KUKA KRL program: vw_Sto_cs_user.src, vw_Sto_cs_user.dat

--- vw_Sto_cs_user.src ---
&ACCESS RVEO
&REL 70
&PARAM DISKPATH = VW_User/Applikation/Vision/SMA
&PARAM TPVW_VERSION = 8.1.8
&PARAM EDITMASK = vw_cgx_user
DEF vw_sto_cs_user( )
;
;*---------------------------------------------*
;* Steinbichler Conzept Solutions GmbH             *
;* Version 1.0.0  / VKRC 4                               *
;* Bearbeitet am:                                          *
;* 20130208  vw_sto_cs_user erstellt                *
;*---------------------------------------------*
;
END
;
GLOBAL DEF STO_CS_Interface(USER_CMD :IN, CMD_SEL :IN,PAR1 :IN,PAR2 :IN, PAR3 :IN,PAR4 :IN,PAR5 :IN,PAR6 :IN)
  DECL VW_USER_CMD USER_CMD
  INT CMD_SEL,PAR1,PAR2,PAR3,PAR4,PAR5,PAR6

  SWITCH PAR1
  ;;FOLD VISIO7
  ;Start Integration VISIO7 durch CS JZ
  ;***********************************************
  ;
  ;***Legende***
	;PAR1 ==> Programmfunktion (1=Bewegung ausfuehren)
	;PAR2 ==> 1=pruefen ob Startpos == AxisRobGst(Home) / 2=nicht pruefen (aus Cell =>2 sonst 1)
	;PAR3 ==> Reserve
	;PAR4 ==> Reserve
	;PAR5 ==> Reserve
	;PAR6 ==> Reserve
	;**************
	;***Interrupts***
	; Interrupt 32 => NOT diZustimm , I_Zustimm()
	; Interrupt 33 => giZyklusCounterIn<>OldZyklusCounterIn , I_Multiplex()
	;**************

CASE 1 ;Bewegung von VISIO7 ausfuehren
 InitVisio () ;Variablen Initialisieren
 PTP $Pos_Act

 OldZyklusCounterIn=giZyklusCounterIn ;auf gleichen Wert setzen um Flanke fuer Interrupt zu bekommen
 INTERRUPT DECL 33 WHEN  giZyklusCounterIn<>OldZyklusCounterIn DO I_Multiplex()
 INTERRUPT ON 33 ;I_Multiplex
 WAIT FOR (OldZyklusCounterIn==giZyklusCounterIn) ; ;auf gleichen Wert warten um Flanke fuer Interrupt zu bekommen
 WAIT SEC 0.15 ;Wartezeit wegen Signalueberschneidung (Falnke Interrupt)
 OldZyklusCounterIn=0 ;mit 0 initialisieren

 IF (PAR2==1) THEN ;pruefen ob Startpos == AxisRobGst(Home)
  bRobGst=IN_AxPOS(AxisRobGst) ;Grundstellung Roboter pruefen Achswerte
  IF NOT bRobGst THEN ; Roboter nicht in Grundtstellung bei Programmeinsprung
   SetProgStatus(203) ;Programmstatus setzen (Legende im SetProgStatus)
   HALT ;ungueltige Startposition (nicht Home)
  ENDIF ; Roboter nicht in Grundtstellung bei Programmeinsprung
 ENDIF ;pruefen ob Startpos == AxisRobGst(Home)
  WAIT FOR bReadComplete ;eimal alle Daten eingelesen, da sonst kein Teachmode gesetzt ist und aus dem Programm gesprungen wird
   REPEAT  ;Onlinefahren ende
      WAIT SEC 0.1 ;Wartezeit wegen CPU-Auslastung
      SetProgStatus(0) ;Programmstatus setzen (Legende im SetProgStatus)

      IF bMoveToPos THEN
         GetSpeed() ;Geschwindigkeitsdaten aus XML auslesen
        IF bErrGetSpeed==FALSE THEN ;kein Fehler Speeddata
         GetPosition() ;Positionsdaten aus XML auslesen
        ENDIF
        bErrGetSpeed=FALSE ;Variable ruecksetzen
      ENDIF

    bRobGst=IN_AxPOS(AxisRobGst) ;Grundstellung Roboter pruefen Achswerte
    IF (bTeachMode==FALSE) AND (bRobGst==FALSE) THEN;teachen beendet, Rob aber nicht in Gst
     SetProgStatus(106) ;Programmstatus setzen (Legende im SetProgStatus)
    ENDIF ;teachen beendet, Rob aber nicht in Gst
   UNTIL (bTeachMode==FALSE) AND (bRobGst==TRUE) ;Onlinefahren ende

    PTP AxisRobGst ;AxisRobGst => entspricht Home in Config.dat
   WAIT SEC 0.0 ;Dummywartezeit wegen Vorlaufstop

   INTERRUPT OFF 33 ;I_Multiplex
    InitVisio () ;Variablen Initialisieren

   DEFAULT
  ENDSWITCH ;von PAR1
  ;***********************************************
  ;Ende Integration VISIO7 durch CS JZ
  ;lokale Unterprogramme am Schluss angehaengt
  ; => DEF InitVisio () ;Variablen Initialisieren
  ; => DEF SetProgStatus(Status :IN)
  ; => DEF GetPosition ()
  ; => DEF GetSpeed()
  ; => DEF MoveToPos()
  ; => DEF I_Zustimm()
  ; => DEF  I_Multiplex()
  ; => DEFFCT  BOOL IN_POS(CHECKPOS :IN)
  ; => DEFFCT  BOOL IN_AxPOS(CHECKPOS :IN)
  ; => DEFFCT INT ByteSwap(nInValue:IN, Lenght:IN, OutSequence:IN, DoFct:IN  )
  ;***********************************************
END
;-----------------------------------------------------------
DEF InitVisio () ;Variablen Initialisieren
 ;Variablen auf Startzuststand Initialisieren
 nProgStatus=0 ;Programmstatus ruecksetzen
 OldZyklusCounterIn=0 ;Multiplexvariable initialisiere
 goZyklusCounterOut=0 ;Ausgang Initialisieren
 bMoveToPos=FALSE ;Auf Position von Visio fahren
 bTeachMode=FALSE ;Teachmode aktiv
 bErrGetSpeed=FALSE ;Fehler in Geschwindigkeitsparameter
 $Timer[nLifeBitTimerNr]=nLifeBitTime ;Timer initialisieren
 $Timer_Stop[nLifeBitTimerNr]=TRUE ;Timer stoppen
 bReadComplete=FALSE ;Merker ruecksetzen
END
;-----------------------------------------------------------
DEF SetProgStatus(Status :IN)
;;FOLD SetProgStatus
   INT Status
   ;====== Legende  Programmstatus=======
   ; 0 => Ready
   ; 1 => Working
   ; 2 => ok (Befehl ausgefuerht)
   ; 10-99 => Zustand
   ; 10 => Robter wird gerade Handgefuehrt
   ;
   ; 100-999 => Fehler
   ; 100 =>
   ; 106 => Teachmode  beendet Roboter aber nicht in Home1 (Teachmode aktivieren undHome1 anfahren)
   ; 116 => anfahren des VisioPunkt durch loslassen der Zustimmtaste abgebrochen
   ; 117 => anfahren des VisioPunkt angewaehlt ohne Zustimmtaste
   ;
   ; 200 => Arbeitsraum-Fehler bei pPosVonVisio
   ; 201 => TURN-Fehler bei pPosVonVisio
   ; 202 => ungueltiger Geschwindigkeitsparameter
   ; 203 => Grundstellungspruefung bei Start TeachMode aktiv => Roboter aber nicht in GST
   ;
   ; 999 => schwerer Fehler Roboterpanel beachten
   ;================================

 IF bKommAktiv THEN ;wenn Kommunikation akitv ist
  WAIT FOR nProgStatusAck==nProgStatus ;Programmstatus Rueckmeldung von Visio
 ENDIF ;wenn Kommunikation akitv ist
 nProgStatus = Status ;Programmstatus setzen

;;ENDFOLD
END
;-----------------------------------------------------------
DEF GetPosition ()

;;FOLD GetPosition
   INTERRUPT DECL 32 WHEN NOT bZustimm DO I_Zustimm()

   IF bZustimm THEN ;wenn Zustimmtaste gedrueckt ist

   SetProgStatus(1) ;Programmstatus setzen (Legende im SetProgStatus)

   ;Positionsdaten wurden bereits im Multiplex-Programm gelesen
   ;Positionsdaten pruefen
   ;E6AXIS  INVERSE (E6POS  POSITION: IN, E6AXIS START_AXIS: IN,				 INT ERR_STATUS: OUT)
   ret=0 ;Variable initialisieren
   APOS1=INVERSE(pPosVonVisio,$Axis_Act,ret)
   IF ret<>0 THEN
    IF ret==2 THEN ;2Arbeitsraum-Fehler bei der math. Trafo-Funktion, d.h. es gibt keine Achswinkel, mit denen die kartesische Zielposition erreicht werden kann
     SetProgStatus(200) ;Programmstatus setzen (Legende im SetProgStatus)
     ELSE ;2
      IF ret==3 THEN ;3 Es gibt zwar Loesungswinkel, aber mit dem gegebenem Turn werden SW-Endschalter verletzt
       SetProgStatus(201) ;Programmstatus setzen (Legende im SetProgStatus)
       ELSE ;3
         HALT ;Roboterposition nicht erreichbar
      ENDIF ;3
    ENDIF ;2
   ELSE ;<>0
   MoveToPos() ;Position anfahren
   ENDIF ;<>0

  ELSE ;wenn Zustimmtaste gedrueckt ist
   SetProgStatus(117) ;Position anfahren gewaehlt aber Zustimmtaste nicht gedrueckt
  ENDIF ;wenn Zustimmtaste gedrueckt ist

;;ENDFOLD
END
;-----------------------------------------------------------
DEF GetSpeed()
;   ;FOLD GetSpeed
   INT Factor,I

   bErrGetSpeed=FALSE ;Variable ruecksetzen

   ; $APO.CDIS
   IF (TeachSpeed.ApoCdis>0) AND (TeachSpeed.ApoCdis<=200) THEN
    IF TeachSpeed.ApoCdis>SpeedLimit.ApoCdis THEN
     TeachSpeed.ApoCdis=SpeedLimit.ApoCdis
    ENDIF
    $APO.CDIS=TeachSpeed.ApoCdis
   ELSE
    SetProgStatus(202) ;Programmstatus setzen (Legende im SetProgStatus)
    User_Msg(2) ;Meldungsausgabe am KCP
    bErrGetSpeed=TRUE ;Variable setzen
   ENDIF

   ; $VEL.CP
   IF (TeachSpeed.VelCp>0) AND (TeachSpeed.VelCp<=2.0) THEN
    IF TeachSpeed.VelCp>SpeedLimit.VelCp THEN
     TeachSpeed.VelCp=SpeedLimit.VelCp
    ENDIF
    $VEL.CP=TeachSpeed.VelCp
   ELSE
    SetProgStatus(202) ;Programmstatus setzen (Legende im SetProgStatus)
    User_Msg(3) ;Meldungsausgabe am KCP
    bErrGetSpeed=TRUE ;Variable setzen
   ENDIF

   ; $ACC.CP
   IF (TeachSpeed.AccCp>0) AND (TeachSpeed.AccCp<=2.3) THEN
    IF TeachSpeed.AccCp>SpeedLimit.AccCp THEN
     TeachSpeed.AccCp=SpeedLimit.AccCp
    ENDIF
    $ACC.CP=TeachSpeed.AccCp
   ELSE
    SetProgStatus(202) ;Programmstatus setzen (Legende im SetProgStatus)
    User_Msg(4) ;Meldungsausgabe am KCP
    bErrGetSpeed=TRUE ;Variable setzen
   ENDIF

   ; $VEL.ORI2
   IF (TeachSpeed.VelOri>0) AND (TeachSpeed.VelOri<=200.0) THEN
    IF TeachSpeed.VelOri>SpeedLimit.VelOri THEN
     TeachSpeed.VelOri=SpeedLimit.VelOri
    ENDIF
    $VEL.ORI1=TeachSpeed.VelOri
    $VEL.ORI2=TeachSpeed.VelOri
   ELSE
    SetProgStatus(202) ;Programmstatus setzen (Legende im SetProgStatus)
    User_Msg(5) ;Meldungsausgabe am KCP
    bErrGetSpeed=TRUE ;Variable setzen
   ENDIF

   ; VELPTP
   ;Factor darf zwischen 0 und 100 liegen
   IF TeachSpeed.VelPtp>SpeedLimit.VelPtp THEN
      TeachSpeed.VelPtp=SpeedLimit.VelPtp
      IF bStopOnError THEN ;bei Fehler halten
       HALT
      ENDIF ;bei Fehler halten
   ENDIF
   IF TeachSpeed.VelPtp<1 THEN ;min 1% Geschwindigkeit
      TeachSpeed.VelPtp=1
      IF bStopOnError THEN ;bei Fehler halten
       HALT
      ENDIF ;bei Fehler halten
   ENDIF
   ;Achsgeschwindigkeiten setzen
   FOR I=1 TO $NUM_AX
      $VEL_AXIS[I]=TeachSpeed.VelPtp
   ENDFOR

   ; ACCPTP
   ;Factor darf zwischen 0 und 100 liegen
   IF TeachSpeed.AccPtp>SpeedLimit.AccPtp THEN
      TeachSpeed.AccPtp=SpeedLimit.AccPtp
   ENDIF
   IF TeachSpeed.AccPtp<1 THEN ;min 1% Beschleunigung
      TeachSpeed.AccPtp=1
   ENDIF
   ;Achsgeschwindigkeiten setzen
   FOR I=1 TO $NUM_AX
      $ACC_AXIS[I]=TeachSpeed.AccPtp
   ENDFOR

   ; $VEL_EXTAX[1]
   ;Factor darf zwischen 0 und 100 liegen
   IF TeachSpeed.VelExtAx1>SpeedLimit.VelExtAx1 THEN
      TeachSpeed.VelExtAx1=SpeedLimit.VelExtAx1
   ENDIF
   IF TeachSpeed.VelExtAx1<1 THEN ;min 1%
      TeachSpeed.VelExtAx1=1
   ENDIF
   ;Achsgeschwindigkeiten setzen
   $VEL_EXTAX[1]=TeachSpeed.VelExtAx1

   ; $VEL_EXTAX[2]
   ;Factor darf zwischen 0 und 100 liegen
   IF TeachSpeed.VelExtAx2>SpeedLimit.VelExtAx2 THEN
      TeachSpeed.VelExtAx2=SpeedLimit.VelExtax2
   ENDIF
   IF TeachSpeed.VelExtAx2<1 THEN ;min 1%
      TeachSpeed.VelExtAx2=1
   ENDIF
   ;Achsgeschwindigkeiten setzen
   $VEL_EXTAX[2]=TeachSpeed.VelExtAx2

;;ENDFOLD
END
;-----------------------------------------------------------
DEF MoveToPos()
   INTERRUPT ON 32 ;Bewegung abbrechen
   WAIT FOR bZustimm ;Zustimmstaste gedrueckt
   IF bMovePTP THEN ;Bewegung ist PTP
      PTP pPosVonVisio ;Punkt anfahren
   ELSE
      LIN pPosVonVisio ;Punkt anfahren
   ENDIF
   Interrupt OFF 32 ;Bewegung abbrechen
   SetProgStatus(2) ;Programmstatus setzen (Legende im SetProgStatus)
END
;-----------------------------------------------------------
DEF I_Zustimm()
   Interrupt OFF 32 ;Bewegung abbrechen
   Brake ;Roboter anhalten
   SetProgStatus(116) ;Programmstatus setzen (Legende im SetProgStatus)
   Resume ;Ruecksprung ins Hauptprogramm
END
;-----------------------------------------------------------
DEF I_Multiplex()
;20130121 JZ => erstellt
;20130125 JZ => neue Signalliste verwendet, Shattendaten erstellt
;29130125 JZ => in VW_USR_R integriert

;bei 5 auf 0 Ruecksetzen, wegen Errorflag bei verpassten Paketen
IF (OldZyklusCounterIn==MultiplexFaktor) OR  ($Timer_Flag[nLifeBitTimerNr]) THEN
 OldZyklusCounterIn=0
 IF $Timer_Flag[nLifeBitTimerNr] THEN
  $Timer[nLifeBitTimerNr]=nLifeBitTime ;Timer initialisieren
  $Timer_Stop[nLifeBitTimerNr]=FALSE ;Timer starten
 ENDIF
ENDIF

IF (ErrorFlag==FALSE) AND (giZyklusCounterIn>1)  AND (giZyklusCounterIn-OldZyklusCounterIn >1) THEN ;Paketverlust
 ErrorFlag=TRUE ;Fehler
 ErrorCounter=ErrorCounter+1 ;Fehlerzaehler hochzaehlen
ENDIF ;Paketverlust

OldZyklusCounterIn=giZyklusCounterIn ;Merker setzen

IF goZyklusCounterOut==giZyklusCounterOutAck THEN ;Im Handhakemodus auf Bestaetigung ZyklusCounterOut warten
goZyklusCounterOut=goZyklusCounterOut+1 ;hochzaehlen
 IF (goZyklusCounterOut>MultiplexFaktor) THEN
  goZyklusCounterOut=1 ;ruecksetzen
 ENDIF
ENDIF

;Am Anfang einer Runde die Schattendaten schreiben
IF goZyklusCounterOut==1 THEN
 ;allgemeine Daten in Schattendaten schreiben
 bSdwDoLifeBit=bLifeBitOld ;
 bSdwDoStopMess=$StopMess ;
 nSdwGoProgStatus=nProgStatus
 nSdwGoRobTimer=$Rob_Timer
 nSdwGoFloatFaktor=nFloatFaktor*10
 ;Positionsdaten in Schattendaten schreiben
 pShadowPosAnVisio=$Pos_Act ;aktuelle Position in Schattendaten speichern
ENDIF

;eine Seite einlesen
IF (giZyklusCounterIn>=1) AND (giZyklusCounterIn<= MultiplexFaktor) THEN
 IF giZyklusCounterIn==1 THEN ;allgemeine Daten
  bSdwDiKommAktiv=diKommAtiv ;
  bSdwDiTeachMode=diTeachMode ;
  bSdwDiMovePTP=diMovePTP ;
  bSdwDiMoveToPos=diMoveToPos ;
  bSdwDiLifeBit=diLifeBit ;
  nSdwGiProgStatusAck=ByteSwap(giProgStatusAck, 16, 21, TRUE) ;
  nSdwGiFloatFaktor=giFloatFaktor*10 ;
  IF nSdwGiFloatFaktor==0 THEN ;ungueltiger Wert wegen Division durch Null
   nSdwGiFloatFaktor=1 ;Wert initialisieren
  ENDIF
 ENDIF ;allgemeine Daten
 IF giZyklusCounterIn==2 THEN ;X/Y/Z
  IF nSdwGiFloatFaktor==0 THEN ;ungueltiger Wert wegen Division durch Null
   nSdwGiFloatFaktor=1 ;Wert initialisieren
  ENDIF
  pShadowPosVonVisio.X=ByteSwap(giPosX, 32, 4321, TRUE)/nSdwGiFloatFaktor
  pShadowPosVonVisio.Y=ByteSwap(giPosY, 32, 4321, TRUE)/nSdwGiFloatFaktor
  pShadowPosVonVisio.Z=ByteSwap(giPosZ, 32, 4321, TRUE)/nSdwGiFloatFaktor
 ENDIF ;X/Y/Z
 IF giZyklusCounterIn==3 THEN ;A/B/C
  IF nSdwGiFloatFaktor==0 THEN ;ungueltiger Wert wegen Division durch Null
   nSdwGiFloatFaktor=1 ;Wert initialisieren
  ENDIF
  pShadowPosVonVisio.A=ByteSwap(giPosA, 32, 4321, TRUE)/nSdwGiFloatFaktor
  pShadowPosVonVisio.B=ByteSwap(giPosB, 32, 4321, TRUE)/nSdwGiFloatFaktor
  pShadowPosVonVisio.C=ByteSwap(giPosC, 32, 4321, TRUE)/nSdwGiFloatFaktor
 ENDIF ;A/B/C
 IF giZyklusCounterIn==4 THEN ;E1/E2/S/T
  IF nSdwGiFloatFaktor==0 THEN ;ungueltiger Wert wegen Division durch Null
   nSdwGiFloatFaktor=1 ;Wert initialisieren
  ENDIF
  pShadowPosVonVisio.E1=ByteSwap(giPosE1, 32, 4321, TRUE)/nSdwGiFloatFaktor
  pShadowPosVonVisio.E2=ByteSwap(giPosE2, 32, 4321, TRUE)/nSdwGiFloatFaktor
  pShadowPosVonVisio.S=giPosS
  pShadowPosVonVisio.T=giPosT ;ByteSwap???
 ENDIF ;E1/E2/S/T
 IF giZyklusCounterIn==5 THEN ;Geschwindigkeitsdaten
  IF nSdwGiFloatFaktor==0 THEN ;ungueltiger Wert wegen Division durch Null
   nSdwGiFloatFaktor=1 ;Wert initialisieren
  ENDIF
  SdwTeachSpeed.ApoCdis=ByteSwap(giApoCdis, 16, 21, TRUE)/100.0
  SdwTeachSpeed.VelCp=ByteSwap(giVelCp, 16, 21, TRUE)/1000.0
  SdwTeachSpeed.AccCp=ByteSwap(giAccCp, 16, 21, TRUE)/100.0
  SdwTeachSpeed.VelOri=ByteSwap(giVelOri, 16, 21, TRUE)
  SdwTeachSpeed.VelPtp=giVelPtp
  SdwTeachSpeed.AccPtp=giAccPtp
  SdwTeachSpeed.VelExtAx1=giVelExtAx1
  SdwTeachSpeed.VelExtAx2=giVelExtAx2
 ENDIF ;Geschwindigkeitsdaten
ENDIF

;eine Seite schreiben
IF (goZyklusCounterOut>=1) AND (goZyklusCounterOut<=MultiplexFaktor) THEN
 IF goZyklusCounterOut==1 THEN ;allgemeine Daten
  I4=$Rob_timer-I3 ;IBN
  I3=$Rob_timer ;IBN
  doLifeBit=bSdwDoLifeBit
  doStopMess=bSdwDoStopMess
  goProgStatus=ByteSwap(nSdwGoProgStatus, 16, 21, TRUE)
  goRobTimer=ByteSwap(nSdwGoRobTimer, 32, 4321, TRUE)
  goFloatFaktor=nSdwGoFloatFaktor/10
 ENDIF ;allgemeine Daten
 IF goZyklusCounterOut==2 THEN ;X/Y/Z
  goPosX=ByteSwap((pShadowPosAnVisio.X*nSdwGoFloatFaktor), 32, 4321, TRUE)
  goPosY=ByteSwap((pShadowPosAnVisio.Y*nSdwGoFloatFaktor), 32, 4321, TRUE)
  goPosZ=ByteSwap((pShadowPosAnVisio.Z*nSdwGoFloatFaktor), 32, 4321, TRUE)
  nGoPosX=goPosX ;IBN
  nGoPosY=goPosY ;IBN
  nGoPosZ=goPosZ ;IBN
 ENDIF ;X/Y/Z
 IF goZyklusCounterOut==3 THEN ;A/B/C
  goPosA=ByteSwap((pShadowPosAnVisio.A*nSdwGoFloatFaktor), 32, 4321, TRUE)
  goPosB=ByteSwap((pShadowPosAnVisio.B*nSdwGoFloatFaktor), 32, 4321, TRUE)
  goPosC=ByteSwap((pShadowPosAnVisio.C*nSdwGoFloatFaktor), 32, 4321, TRUE)
  nGoPosA=goPosA ;IBN
  nGoPosB=goPosB ;IBN
  nGoPosC=goPosC ;IBN
 ENDIF ;A/B/C
 IF goZyklusCounterOut==4 THEN ;E1/E2/S/T
  goPosE1=ByteSwap((pShadowPosAnVisio.E1*nSdwGoFloatFaktor), 32, 4321, TRUE)
  goPosE2=ByteSwap((pShadowPosAnVisio.E2*nSdwGoFloatFaktor), 32, 4321, TRUE)
  goPosS=pShadowPosAnVisio.S
  goPosT=pShadowPosAnVisio.T
  goPosT2=0 ;ReserveTurn auf 0 initialisieren
  goPosT3=0 ;ReserveTurn auf 0 initialisieren
  nGoPosE1=goPosE1 ;IBN
  nGoPosE2=goPosE2 ;IBN
  nGoPosS=goPosS ;IBN
  nGoPosT=goPosT ;IBN
 ENDIF ;E1/E2/S/T
 IF goZyklusCounterOut==5 THEN ;Reserve
  ;nicht belegt
 ENDIF ;
ENDIF

;Am Ende einer Runde die Schattendaten uebernehmen
IF (ErrorFlag==FALSE) AND (giZyklusCounterIn==MultiplexFaktor) THEN
  bKommAktiv=bSdwDiKommAktiv ;
  bTeachMode=bSdwDiTeachMode ;
  bMovePTP=bSdwDiMovePTP ;
  bMoveToPos=bSdwDiMoveToPos ;
  bLifeBit=bSdwDiLifeBit ;
  nProgStatusAck=nSdwGiProgStatusAck ;
  ;nSdwGiFloatFaktor ;wird nur im Multiplexbereich benoetigt
  pPosVonVisio=pShadowPosVonVisio ;Positionsdaten uebergeben
  TeachSpeed.ApoCdis =SdwTeachSpeed.ApoCdis
  TeachSpeed.VelCp =SdwTeachSpeed.VelCp
  TeachSpeed.AccPtp =SdwTeachSpeed.AccPtp
  TeachSpeed.VelOri =SdwTeachSpeed.VelOri
  TeachSpeed.VelPtp =SdwTeachSpeed.VelPtp
  TeachSpeed.AccPtp =SdwTeachSpeed.AccPtp
  TeachSpeed.VelExtAx1 =SdwTeachSpeed.VelExtAx1
  TeachSpeed.VelExtAx2 =SdwTeachSpeed.VelExtAx2
  ;Lifebit
  IF bLifeBit==bLifeBitOld THEN ;LifeBit vergleichen
   bLifeBitOld=NOT bLifeBitOld ;Lifebit negieren
   I2=$Rob_timer-I1 ;IBN
   I1=$Rob_timer ;IBN
   $Timer[nLifeBitTimerNr]=nLifeBitTime ;Timer initialisieren
   $Timer_Stop[nLifeBitTimerNr]=FALSE ;Timer starten
  ENDIF ;LifeBit vergleichen
 bReadComplete=TRUE ;1 Datensatz komplett gelesen
ENDIF

IF ErrorFlag AND (giZyklusCounterIn==1) THEN
 ErrorFlag=FALSE ;Flag ruecksetzen
ENDIF

;Spiegeln fuer die Gegenseite
goZyklusCounterInAck=giZyklusCounterIn

END
;-----------------------------------------------------------
;FOLD Position pruefen
DEFFCT  BOOL IN_POS(CHECKPOS :IN)
DECL E6POS CHECKPOS
DECL BOOL B_IN_POS
B_IN_POS=TRUE
IF (CHECKPOS.X<$POS_ACT.X-TolTrans) OR (CHECKPOS.X>$POS_ACT.X+TolTrans) THEN
 B_IN_POS=FALSE
ENDIF
IF (CHECKPOS.Y<$POS_ACT.Y-TolTrans) OR (CHECKPOS.Y>$POS_ACT.Y+TolTrans) THEN
 B_IN_POS=FALSE
ENDIF
IF (CHECKPOS.Z<$POS_ACT.Z-TolTrans) OR (CHECKPOS.Z>$POS_ACT.Z+TolTrans) THEN
 B_IN_POS=FALSE
ENDIF
IF (CHECKPOS.A<$POS_ACT.A-TolRot) OR (CHECKPOS.A>$POS_ACT.A+TolRot) THEN
 B_IN_POS=FALSE
ENDIF
IF (CHECKPOS.B<$POS_ACT.B-TolRot) OR (CHECKPOS.B>$POS_ACT.B+TolRot) THEN
 B_IN_POS=FALSE
ENDIF
IF (CHECKPOS.C<$POS_ACT.C-TolRot) OR (CHECKPOS.C>$POS_ACT.C+TolRot) THEN
 B_IN_POS=FALSE
ENDIF
IF (CHECKPOS.E1<$POS_ACT.E1-TolRot) OR (CHECKPOS.E1>$POS_ACT.E1+TolRot) THEN
 B_IN_POS=FALSE
ENDIF
IF (CHECKPOS.E2<$POS_ACT.E2-TolRot) OR (CHECKPOS.E2>$POS_ACT.E2+TolRot) THEN
 B_IN_POS=FALSE
ENDIF
RETURN  (B_IN_POS)
ENDFCT ;Function IN_POS
;ENDFOLD
;-----------------------------------------------------------
;FOLD Achsposition pruefen
DEFFCT  BOOL IN_AxPOS(CHECKPOS :IN)
DECL E6AXIS CHECKPOS
DECL BOOL B_IN_POS
B_IN_POS=TRUE
IF (CHECKPOS.A1<$AXIS_ACT.A1-TolRot) OR (CHECKPOS.A1>$AXIS_ACT.A1+TolRot) THEN
 B_IN_POS=FALSE
ENDIF
IF (CHECKPOS.A2<$AXIS_ACT.A2-TolRot) OR (CHECKPOS.A2>$AXIS_ACT.A2+TolRot) THEN
 B_IN_POS=FALSE
ENDIF
IF (CHECKPOS.A3<$AXIS_ACT.A3-TolRot) OR (CHECKPOS.A3>$AXIS_ACT.A3+TolRot) THEN
 B_IN_POS=FALSE
ENDIF
IF (CHECKPOS.A4<$AXIS_ACT.A4-TolRot) OR (CHECKPOS.A4>$AXIS_ACT.A4+TolRot) THEN
 B_IN_POS=FALSE
ENDIF
IF (CHECKPOS.A5<$AXIS_ACT.A5-TolRot) OR (CHECKPOS.A5>$AXIS_ACT.A5+TolRot) THEN
 B_IN_POS=FALSE
ENDIF
IF (CHECKPOS.A6<$AXIS_ACT.A6-TolRot) OR (CHECKPOS.A6>$AXIS_ACT.A6+TolRot) THEN
 B_IN_POS=FALSE
ENDIF
IF (CHECKPOS.E1<$AXIS_ACT.E1-TolRot) OR (CHECKPOS.E1>$AXIS_ACT.E1+TolRot) THEN
 B_IN_POS=FALSE
ENDIF
IF (CHECKPOS.E2<$AXIS_ACT.E2-TolRot) OR (CHECKPOS.E2>$AXIS_ACT.E2+TolRot) THEN
 B_IN_POS=FALSE
ENDIF
RETURN  (B_IN_POS)
ENDFCT ;Function IN_POS
;ENDFOLD
;-----------------------------------------------------------
DEFFCT INT ByteSwap(nInValue:IN, Lenght:IN, OutSequence:IN, DoFct:IN  )

INT Result ;Ergebnis der Funktion
INT nInValue ;Eingangswert der umgewandelt werden soll
INT Lenght ;Bitanzahl des Eingangswertes (16 / 32)
BOOL DoFct ;ob die Funktion ausgefuehrt werden soll
INT SwapByte1, SwapByte2, SwapByte3, SwapByte4 ;Rechenbytes
INT OutSequence ;Reihenfolge in der die Bytes ausgegeben werden (z.B. Eingang 1,2,3,4 => Ausgang 4,3,2,1)
BOOL HiBit ;fuer Auswertung negative Zahl

;#######################################
;Wenn allgemein diese Funktion ausgeschaltet werden soll hier die Variable setzen
;DoFct=FALSE
;#######################################

IF DoFct THEN ;Berechnungen ausfuehren
 SwapByte1='B00000000' ;Initialisieren
 SwapByte2='B00000000' ;Initialisieren
 SwapByte3='B00000000' ;Initialisieren
 SwapByte4='B00000000' ;Initialisieren
 SWITCH Lenght
 ;----------------------------------------
  CASE 16 ;16 Bit Eingang
   SWITCH OutSequence ;Reihenfolge der Bytes
   ;==================================
    CASE 21
     SwapByte1= nInValue B_AND 'B1111111100000000'
     SwapByte2= nInValue B_AND 'B0000000011111111'
     SwapByte1=SwapByte1/256 ;Byte um 1 nach hinten schieben (2=>1)
     SwapByte2=SwapByte2*256 ;Byte um 1 nach vorn schieben (1=>2)
     Result=SwapByte1+SwapByte2 ;SwapBytes addieren
   ;==================================
    DEFAULT ;Reihenfolge der Bytes
     User_Msg(6) ;Meldungsausgabe am KCP
    ENDSWITCH ;Reihenfolge der Bytes
 ;----------------------------------------
  CASE 32 ;32 Bit Eingang
   SWITCH OutSequence ;Reihenfolge der Bytes
   ;==================================
    CASE 4321
     SwapByte1= nInValue B_AND 'B01111111000000000000000000000000'
     HiBit = (nInValue B_AND 'B10000000000000000000000000000000' <>0) ;abfangen wegen Negativer Zahlen (an Ende +128 rechnen)
     SwapByte2= nInValue B_AND 'B00000000111111110000000000000000'
     SwapByte3= nInValue B_AND 'B00000000000000001111111100000000'
     SwapByte4= nInValue B_AND 'B00000000000000000000000011111111'
     SwapByte1=(((SwapByte1/256)/256)/256) ;Byte um 3 nach hinten schieben (4=>1)
     SwapByte2=SwapByte2/256 ;Byte um 1 nach hinten schieben (3=>2)
     SwapByte3=SwapByte3*256 ;Byte um 1 nach vorn schieben (2=>3)
     SwapByte4=(((SwapByte4*256)*256)*256) ;Byte um 3 nach vorn schieben (1=>4)
     IF HiBit THEN
      Result=SwapByte1+SwapByte2+SwapByte3+SwapByte4+128 ;SwapBytes addieren und 128 hinzuzaehlen wegen Negativzahl
     ELSE
      Result=SwapByte1+SwapByte2+SwapByte3+SwapByte4 ;SwapBytes addieren
     ENDIF
   ;==================================
    DEFAULT ;Reihenfolge der Bytes
     User_Msg(7) ;Meldungsausgabe am KCP
    ENDSWITCH ;Reihenfolge der Bytes
 ;----------------------------------------
  DEFAULT ;BitZahl
   User_Msg(8) ;Meldungsausgabe am KCP
 ENDSWITCH ;BitZahl

ELSE ;Berechnungen ausfuehren
 Result=nInValue ;Rueckgabewert aus Eingabewert setzen bei Nichtberechnung
ENDIF  ;Berechnungen ausfuehren

RETURN(Result) ;Ergebnis von Funktion Uebergeben
ENDFCT

;-----------------------------------------------------------
DEF User_Msg(MyMsgNr:IN )

 ;FOLD Versionslegende

 ;ENDFOLD
;aktuelle Version: V1.0

DECL KrlMsg_T My_Meldung
DECL KrlMsgPar_T My_Parameter[3]
DECL KrlMsgOpt_T My_Option
DECL KrlMsgDlgSK_T My_SK[7]
int Result, MyMsgNr, Answer
;BOOL Clear_Ok ;Global in $Config.dat
INT MsgHandle[200] ;Handle der Meldung

;---------------------------------------------------
;#notify => Hinweismeldung
;                 -(nur mit Quitt / Alles Quitt)
;#state => Zustandsmeldung
;                -(von Programm aus löschbar)
;#quit => Quittiermeldung
;              -(Quitt / Alles Quitt mit rueckmeldung zum Programm)
;#waiting => Wartemeldung
;                  -(Simuliere oder auf Programmbedingung warten)
;---------------------------------------------------

;alle Mledungen loeschen
;Clear_OK = Clear_KrlMsg(-99) ; Meldungen im Puffer zurueck nehmen
IF bShowUserMsg THEN ;Meldungen anzeigen
SWITCH MyMsgNr
;---------------------------------------------------
 CASE 1 ;
  My_Meldung = {Modul[] "STO-CS", Nr 000, Msg_txt[] "fehlerhafte Gruppennummer uebergeben"}
  My_Meldung.Nr = MyMsgNr
  My_Option = {VL_Stop True, Clear_P_Reset True, Log_To_DB True}
  MsgHandle[MyMsgNr] = Set_KrlMsg(#state, My_Meldung, My_Parameter[], My_Option)
;---------------------------------------------------
 CASE 2 ;
  My_Meldung = {Modul[] "STO-CS", Nr 000, Msg_txt[] "TeachSpeed.ApoCdis => Wert ungueltig"}
  My_Meldung.Nr = MyMsgNr
  My_Option = {VL_Stop True, Clear_P_Reset True, Log_To_DB True}
  MsgHandle[MyMsgNr] = Set_KrlMsg(#state, My_Meldung, My_Parameter[], My_Option)
;---------------------------------------------------
 CASE 3 ;
  My_Meldung = {Modul[] "STO-CS", Nr 000, Msg_txt[] "TeachSpeed.VelCp => Wert ungueltig"}
  My_Meldung.Nr = MyMsgNr
  My_Option = {VL_Stop True, Clear_P_Reset True, Log_To_DB True}
  MsgHandle[MyMsgNr] = Set_KrlMsg(#state, My_Meldung, My_Parameter[], My_Option)
;---------------------------------------------------
 CASE 4 ;
  My_Meldung = {Modul[] "STO-CS", Nr 000, Msg_txt[] "TeachSpeed.AccCp => Wert ungueltig"}
  My_Meldung.Nr = MyMsgNr
  My_Option = {VL_Stop True, Clear_P_Reset True, Log_To_DB True}
  MsgHandle[MyMsgNr] = Set_KrlMsg(#state, My_Meldung, My_Parameter[], My_Option)
;---------------------------------------------------
 CASE 5 ;
  My_Meldung = {Modul[] "STO-CS", Nr 000, Msg_txt[] "TeachSpeed.VelOri => Wert ungueltig"}
  My_Meldung.Nr = MyMsgNr
  My_Option = {VL_Stop True, Clear_P_Reset True, Log_To_DB True}
  MsgHandle[MyMsgNr] = Set_KrlMsg(#state, My_Meldung, My_Parameter[], My_Option)
;---------------------------------------------------
 CASE 6 ;
  My_Meldung = {Modul[] "STO-CS", Nr 000, Msg_txt[] "OutSequence 16Bit Eingabe ByteSwap nicht definiert!"}
  My_Meldung.Nr = MyMsgNr
  My_Option = {VL_Stop True, Clear_P_Reset True, Log_To_DB True}
  MsgHandle[MyMsgNr] = Set_KrlMsg(#state, My_Meldung, My_Parameter[], My_Option)
;---------------------------------------------------
 CASE 7 ;
  My_Meldung = {Modul[] "STO-CS", Nr 000, Msg_txt[] "OutSequence 32Bit Eingabe ByteSwap nicht definiert!"}
  My_Meldung.Nr = MyMsgNr
  My_Option = {VL_Stop True, Clear_P_Reset True, Log_To_DB True}
  MsgHandle[MyMsgNr] = Set_KrlMsg(#state, My_Meldung, My_Parameter[], My_Option)
;---------------------------------------------------
 CASE 8 ;
  My_Meldung = {Modul[] "STO-CS", Nr 000, Msg_txt[] "Eingabe Bitlaenge ByteSwap unbekannt!"}
  My_Meldung.Nr = MyMsgNr
  My_Option = {VL_Stop True, Clear_P_Reset True, Log_To_DB True}
  MsgHandle[MyMsgNr] = Set_KrlMsg(#state, My_Meldung, My_Parameter[], My_Option)
;---------------------------------------------------
	CASE 151 ;
		My_Meldung = {Modul[] "STO-CS", Nr 000, Msg_txt[] "Teachmode beendet, Teachmode aktivieren und Roboter in Grundstellung bringen"}
    My_Meldung.Nr = MyMsgNr
		My_Option = {VL_Stop True, Clear_P_Reset True, Clear_P_SAW True, Log_To_DB False}
		MsgHandle[MyMsgNr] = Set_KrlMsg(#Quit, My_Meldung, My_Parameter[], My_Option)
	 WHILE (Exists_KrlMsg(MsgHandle[MyMsgNr])) ;warten bis der Anwender quittiert hat
			WAIT SEC 0.1
		ENDWHILE
	;---------------------------------------------------
DEFAULT
  My_Meldung = {Modul[] "STO-CS", Nr 000, Msg_txt[] "kein Meldetext vorhanden"}
  My_Meldung.Nr = MyMsgNr
  My_Option = {VL_Stop True, Clear_P_Reset True, Log_To_DB False}
  MsgHandle[MyMsgNr] = Set_KrlMsg(#State, My_Meldung, My_Parameter[], My_Option)
		WHILE (Exists_KrlMsg(MsgHandle[MyMsgNr])) ;warten bis der Anwender quittiert hat
			WAIT SEC 0.1
		ENDWHILE
  ;WAIT FOR FALSE
ENDSWITCH
ENDIF ;Meldungen anzeigen

END
;-----------------------------------------------------------
GLOBAL DEF STO_CS_SPS ()
;*** Zusatz für Teachmode mit VISIO7 (CS JZ) ***
 IF $Timer_Flag[nLifeBitTimerNr] THEN ;Timeout Lifebit
  bZustimm=FALSE ;Zustimmtaste ruecksetzen um Bewegung anzubrechen
 ELSE ;kein TimeOut
  bZustimm=diZustimm ;Uebergabe, da bei Busfehler und anstehendem Signal trotzdem gestoppt werden soll
 ENDIF ;Timeout LifeBit
;*** ENDE ****
END

--- vw_Sto_cs_user.dat ---
&ACCESS  RV
&PARAM DISKPATH = VW_User/Applikation/Vision/SMA
&PARAM EDITMASK = vw_cgx_user
&PARAM TPVW_VERSION = 8.1.8
&REL 69
DEFDAT  vw_Sto_cs_user PUBLIC
;
;FOLD STO_CS
;
;*---------------------------------------------*
;* Steinbichler CS GmbH                        *
;*                                             *
;* Bearbeitet am:                              *
;* 20130208 JZ                                 *
;*     vw_sto_cs_user  erstellt                *
;* 20151219 MBA                                *
;*     b_zustimm entfernt                      *
;*---------------------------------------------*
;
GLOBAL BOOL B_MIT_STO_CS=TRUE

INT I1=10717152
INT I2=3311112
INT I3=10721412
INT I4=88

;Allgemeine Variablen
BOOL bReadComplete=FALSE ;Merker 1 Zyklus komplett gelesen
;BOOL bErrGetSpeed=FALSE ;Fehler in Geschwindigkeitsparameter
BOOL bKommAktiv=FALSE ;Kommunikation mit Visio7 aktiv
BOOL bMoveToPos=FALSE ;Auf Position von Visio fahren
INT nProgStatusAck=0 ;Quittierung Programmstatus von Visio
INT nProgStatus=0 ;aktueller Programmstatus
;INT nRobTimer=0 ;Timestamp 1Inc=2ms
;in Config.dat ;BOOL bZustimm=TRUE ;Zustimmtaste
BOOL bMovePTP=FALSE ;Bewegung als PTP(TRUE) oder LIN(FALSE) ausfuehren
BOOL bTeachMode=FALSE ;Teachmode aktiv
BOOL bLifeBit=FALSE ;Lifebit zu Visio7
BOOL bLifeBitOld=TRUE ;Lifebit zu Visio7
GLOBAL BOOL bShowUserMsg=TRUE ;Meldungen am KCP anzeigen

;Allgemeine E/A
DECL E6AXIS APOS1={A1 8.13010216,A2 -82.4998856,A3 76.0127487,A4 269.075317,A5 98.0776978,A6 83.4475708,E1 0.0,E2 0.0,E3 0.0,E4 0.0,E5 0.0,E6 0.0} ;Achspos pPosVonVosio nach Inverse
;DECL E6AXIS APOS1={A1 0.969305158,A2 -145.691193,A3 140.448578,A4 -0.00214473042,A5 -106.031944,A6 -0.756430626,E1 0.000104831379,E2 0.000104831379,E3 0.0,E4 0.0,E5 0.0,E6 0.0} ;Achspos pPosVonVosio nach Inverse
INT ret=0 ;Returnwert aus Inverse-Funktion zur kontrolle ob pPosVonVisio gueltige Position ist
BOOL bRobGst=TRUE ;Roboter in Grundstellung wegen Teachmode beenden
REAL TolTrans=10.0 ;Translatorische Kartesiche Toleranz bei Gst-Pruefung in mm
REAL TolRot=2.0 ;Rotatorische Kartesiche Tolleranz bei Gst-Pruefung  in Grad

BOOL bErrGetSpeed=FALSE ;Fehler in Geschwindigkeitsparameter
BOOL bStopOnError=FALSE ;im Fehlerfall anhalten (IBN)

;Timereinstellungen
GLOBAL INT nLifeBitTimerNr=4 ;Nummer des verwendeten Timers LifeBitueberwachung
GLOBAL INT nLifeBitTime=-1000 ;Lifebit max. Zeit fuer Wechsel

;Positionsdaten
DECL GLOBAL E6AXIS AxisRobGst={A1 8.13010216,A2 -82.4998856,A3 76.0127487,A4 269.075317,A5 98.0776978,A6 83.4475708,E1 0.0,E2 0.0,E3 0.0,E4 0.0,E5 0.0,E6 0.0}
;GLOBAL DECL E6POS PosRobGst={X 732.678284,Y -12.4045916,Z 1751.1825,A -0.158198372,B -21.2726555,C -0.292230427,S 'B0110',T 'B00111010',E1 0.000104831379,E2 0.000104831379,E3 0.0,E4 0.0,E5 0.0,E6 0.0} ;Positionsdaten an Visio

GLOBAL INT OldZyklusCounterIn=0 ;
BOOL ErrorFlag=FALSE ; Fehler festgestellt
INT ErrorCounter=5 ; Fehlerzaehler

;INT ZyklusCounterIn=0 ; jetzt Signalvereinbarung (Eingaenge)
INT MultiplexFaktor=5 ;Antahl der gemuxten Seiten
INT nFloatFaktor=10 ;(Umrechnungsfaktor = wert *10)
;INT ZyklusCounterOut=1 ; ; jetzt Signalvereinbarung (Ausgaenge)

;Geschwindigkeitsdaten
STRUC SpeedVar REAL ApoCdis,VelOri,INT VelPtp,AccPtp,REAL VelCp,AccCp,INT VelExtAx1,VelExtAx2
DECL SpeedVar TeachSpeed={ApoCdis 0.0,VelOri 0.0,VelPtp 0,AccPtp 0,VelCp 0.0,AccCp 0.300000012,VelExtAx1 0,VelExtAx2 0} ;Speedvar bei Teachmode
DECL SpeedVar SdwTeachSpeed={ApoCdis 0.0,VelOri 0.0,VelPtp 0,AccPtp 0,VelCp 0.0,AccCp 0.0,VelExtAx1 0,VelExtAx2 0} ;Speedvar bei Teachmode
DECL SpeedVar SpeedLimit={ApoCdis 100.0,VelOri 30.0,VelPtp 10,AccPtp 50,VelCp 0.300000012,AccCp 0.300000012,VelExtAx1 20,VelExtAx2 20} ;Speedvar bei Teachmode

;Schattendaten von Visio
DECL E6POS pShadowPosVonVisio={X 0.0,Y 0.0,Z 0.0,A 0.0,B 0.0,C 0.0,S 0,T 0,E1 0.0,E2 0.0,E3 0.0,E4 0.0,E5 0.0,E6 0.0} ;Positiondaten von Visio
BOOL bSdwDiKommAktiv=FALSE ;
BOOL bSdwDiTeachMode=FALSE ;
BOOL bSdwDiMovePTP=FALSE ;
BOOL bSdwDiMoveToPos=FALSE ;
BOOL bSdwDiLifeBit=FALSE ;
INT nSdwGiProgStatusAck=0 ;
INT nSdwGiFloatFaktor=1 ;

DECL E6POS pPosVonVisio={X 0.0,Y 0.0,Z 0.0,A 0.0,B 0.0,C 0.0,S 0,T 0,E1 0.0,E2 0.0,E3 0.0,E4 0.0,E5 0.0,E6 0.0} ;Positiondaten von Visio

;Schattendaten an Visio
DECL E6POS pShadowPosAnVisio={X 1680.0,Y 4.71258772E-06,Z 1910.0,A 0.0,B 90.0,C -90.0,S 'B0010',T 'B0010',E1 0.0,E2 0.0,E3 0.0,E4 0.0,E5 0.0,E6 0.0} ;Positiondaten von Visio
BOOL bSdwDoLifeBit=TRUE ;Schatten-Lifebit
BOOL bSdwDoStopMess=FALSE ;
INT nSdwGoProgStatus=0 ;
INT nSdwGoRobTimer=10721411 ;
INT nSdwGoFloatFaktor=100 ;

;Datenbereich declarieren
;Fester Datenbereich Eingaenge
SIGNAL giZyklusCounterIn $IN[1953]  TO $IN[1960] ; Multiplexzyklus (aktuelle MUX-Seite von VISIO) 8Bit
SIGNAL giZyklusCounterOutAck $IN[1961]  TO $IN[1968] ;ACK (aktuelle MUX-Seite von VISIO als Handshake) 8Bit
;Global in Config.dat angelegt wegen Usr_S;SIGNAL diZustimm $IN[1969] ; Zustimmtaste von VISIO
SIGNAL diContinue $IN[1970] ;Messung beendet => weiterfahrt

;Fester Datenbereich Ausgaenge
SIGNAL goZyklusCounterOut $OUT[1953]  TO $OUT[1960] ; Multiplexzyklus (aktuelle MUX-Seite an VISIO) 8Bit
SIGNAL goZyklusCounterInAck $OUT[1961]  TO $OUT[1968] ;ACK (aktuelle MUX-Seite an VISIO als Handshake) 8Bit
;wird als BinOut konfiguriert;SIGNAL goProgChecksum $OUT[1969]  TO $OUT[1984] ;Programmchecksumme 16Bit
SIGNAL doPosReached $OUT[1985] ;Roboter ist in Messposition

;Multiplexter Datenbereich Eingaenge (von VISIO)
;Seite 1
SIGNAL diKommAtiv $IN[2017] ;Kommunikation aktiv
SIGNAL diTeachMode $IN[2018] ;Teachmode aktiv
SIGNAL diMovePTP $IN[2019] ; ;Bewegung als PTP(TRUE) oder LIN(FALSE) ausfuehren
SIGNAL diMoveToPos $IN[2020] ;Position anfahren start
SIGNAL diLifeBit $IN[2021] ;Lebensbit
SIGNAL giProgStatusAck $IN[2033]  TO $IN[2048] ;Programmstatus Quittierung 16Bit
SIGNAL giFloatFaktor $IN[2049]  TO $IN[2056] ;Floatfaktor Positionsdaten (Umrechnungsfaktor = wert *10) 8Bit
;Seite 2
SIGNAL giPosX $IN[2017]  TO $IN[2048] ;32Bit ProfiNet (Multiplex)
SIGNAL giPosY $IN[2049]  TO $IN[2080] ;32Bit ProfiNet (Multiplex)
SIGNAL giPosZ $IN[2081]  TO $IN[2112] ;32Bit ProfiNet (Multiplex)
;Seite 3
SIGNAL giPosA $IN[2017]  TO $IN[2048] ;32Bit ProfiNet (Multiplex)
SIGNAL giPosB $IN[2049]  TO $IN[2080] ;32Bit ProfiNet (Multiplex)
SIGNAL giPosC $IN[2081]  TO $IN[2112] ;32Bit ProfiNet (Multiplex)
;Seite 4
SIGNAL giPosE1 $IN[2017]  TO $IN[2048] ;32Bit ProfiNet (Multiplex)
SIGNAL giPosE2 $IN[2049]  TO $IN[2080] ;32Bit ProfiNet (Multiplex)
SIGNAL giPosS $IN[2081]  TO $IN[2088] ;8Bit ProfiNet (Multiplex)
SIGNAL giPosT $IN[2089]  TO $IN[2096] ;8Bit ProfiNet (Multiplex)
SIGNAL giPosT2 $IN[2097]  TO $IN[2104] ;8Bit ProfiNet (Multiplex) ReserveTurn
SIGNAL giPosT3 $IN[2105]  TO $IN[2112] ;8Bit ProfiNet (Multiplex) ReserveTurn
;Seite 5
SIGNAL giApoCdis $IN[2017]  TO $IN[2032] ;16Bit ProfiNet (Multiplex)
SIGNAL giVelCp $IN[2033]  TO $IN[2048] ;16Bit ProfiNet (Multiplex)
SIGNAL giAccCp $IN[2049]  TO $IN[2064] ;16Bit ProfiNet (Multiplex)
SIGNAL giVelOri $IN[2065]  TO $IN[2080] ;16Bit ProfiNet (Multiplex)
SIGNAL giVelPtp $IN[2081]  TO $IN[2088] ;8Bit ProfiNet (Multiplex)
SIGNAL giAccPtp $IN[2089]  TO $IN[2096] ;8Bit ProfiNet (Multiplex)
SIGNAL giVelExtAx1 $IN[2097]  TO $IN[2104] ;8Bit ProfiNet (Multiplex)
SIGNAL giVelExtAx2 $IN[2105]  TO $IN[2112] ;8Bit ProfiNet (Multiplex)

;Multiplexter Datenbereich Ausgaenge (an VISIO)
;Seite 1
SIGNAL doLifeBit $OUT[2017] ;Lebensbit
SIGNAL doStopMess $OUT[2018] ;Fehler
SIGNAL goProgStatus $OUT[2033]  TO $OUT[2048] ;Programmstatus 16Bit
SIGNAL goRobTimer $OUT[2049]  TO $OUT[2080] ;Robotertimer 32Bit
SIGNAL goFloatFaktor $OUT[2081]  TO $OUT[2088] ;;Floatfaktor Positionsdaten (Umrechnungsfaktor = wert *10) 8Bit
;Seite 2
SIGNAL goPosX $OUT[2017]  TO $OUT[2048] ;32Bit ProfiNet (Multiplex)
SIGNAL goPosY $OUT[2049]  TO $OUT[2080] ;32Bit ProfiNet (Multiplex)
SIGNAL goPosZ $OUT[2081]  TO $OUT[2112] ;32Bit ProfiNet (Multiplex)
;Seite 3
SIGNAL goPosA $OUT[2017]  TO $OUT[2048] ;32Bit ProfiNet (Multiplex)
SIGNAL goPosB $OUT[2049]  TO $OUT[2080] ;32Bit ProfiNet (Multiplex)
SIGNAL goPosC $OUT[2081]  TO $OUT[2112] ;32Bit ProfiNet (Multiplex)
;Seite 4
SIGNAL goPosE1 $OUT[2017]  TO $OUT[2048] ;32Bit ProfiNet (Multiplex)
SIGNAL goPosE2 $OUT[2049]  TO $OUT[2080] ;32Bit ProfiNet (Multiplex)
SIGNAL goPosS $OUT[2081]  TO $OUT[2088] ;8Bit ProfiNet (Multiplex)
SIGNAL goPosT $OUT[2089]  TO $OUT[2096] ;8Bit ProfiNet (Multiplex)
SIGNAL goPosT2 $OUT[2097]  TO $OUT[2104] ;8Bit ProfiNet (Multiplex) ReserveTurn
SIGNAL goPosT3 $OUT[2105]  TO $OUT[2112] ;8Bit ProfiNet (Multiplex) ReserveTurn
;Seite 5
;RESERVE

;Kontrollvariablen zur IBN
INT nGoPosX='B01000000100100000000001000000000'
INT nGoPosY='B0000'
INT nGoPosZ='B00011000111010100000001000000000'
INT nGoPosA='B0000'
INT nGoPosB='B00101000001000110000000000000000'
INT nGoPosC='B11011000110111001111111111111111'
INT nGoPosE1='B0000'
INT nGoPosE2='B0000'
INT nGoPosS='B0010'
INT nGoPosT='B0010'

;
;ENDFOLD
ENDDAT
